PROGRAM P_MotionSup
VAR
END_VAR

END_PROGRAM

(* stored: Version 1.1.0.1, ProductVersion 3.1.4020.12
   POU P_MotionSup: Id {a34595bb-b6ff-449d-b539-c9e2760a9a1c}, SpecialFunc None *)
